// LS Electric XG5000 project: 과년65_2
// PLC NewPLC
// module base 0 slot 0: 입출력 모듈:XBC-DR20S (DC 24V 입력 12점, 릴레이 출력 8점)

PROGRAM NewProgram (task: 스캔 프로그램)

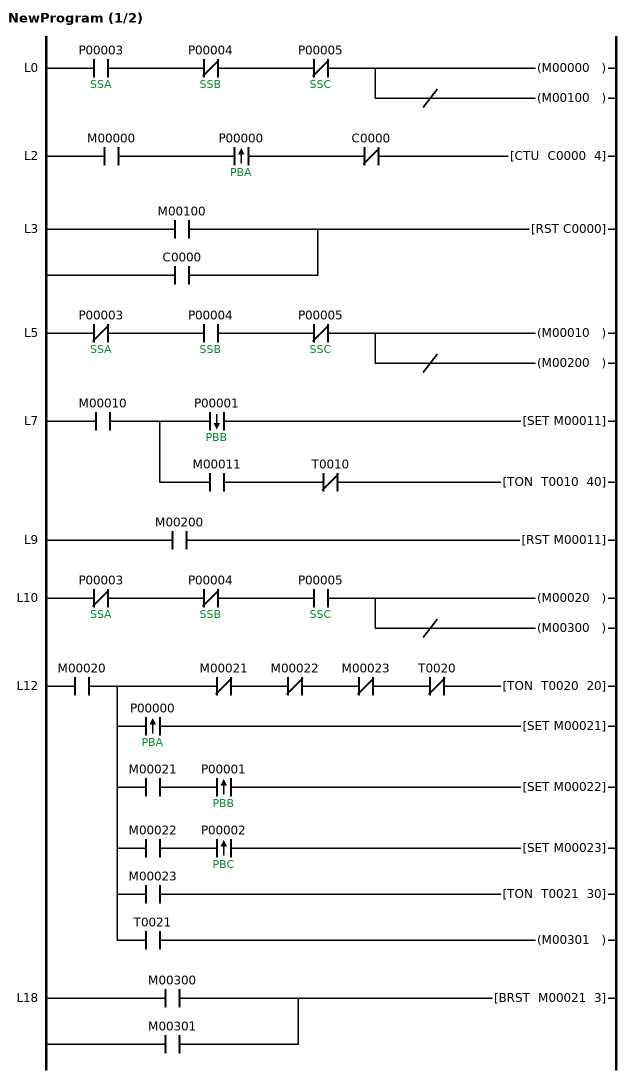
; L0
LOAD      P00003	// SSA
AND NOT   P00004	// SSB
AND NOT   P00005	// SSC
OUT       M00000
NOT
OUT       M00100
; L2
LOAD      M00000
ANDP      P00000	// PBA
AND NOT   C0000
CTU       C0000 4
; L3
LOAD      M00100
OR        C0000
RST       C0000
; L5
LOAD NOT  P00003	// SSA
AND       P00004	// SSB
AND NOT   P00005	// SSC
OUT       M00010
NOT
OUT       M00200
; L7
LOAD      M00010
MPUSH
ANDN      P00001	// PBB
SET       M00011
MPOP
AND       M00011
AND NOT   T0010
TON       T0010 40
; L9
LOAD      M00200
RST       M00011
; L10
LOAD NOT  P00003	// SSA
AND NOT   P00004	// SSB
AND       P00005	// SSC
OUT       M00020
NOT
OUT       M00300
; L12
LOAD      M00020
MPUSH
AND NOT   M00021
AND NOT   M00022
AND NOT   M00023
AND NOT   T0020
TON       T0020 20
MLOAD
ANDP      P00000	// PBA
SET       M00021
MLOAD
AND       M00021
ANDP      P00001	// PBB
SET       M00022
MLOAD
AND       M00022
ANDP      P00002	// PBC
SET       M00023
MLOAD
AND       M00023
TON       T0021 30
MPOP
AND       T0021
OUT       M00301
; L18
LOAD      M00300
OR        M00301
BRST      M00021 3

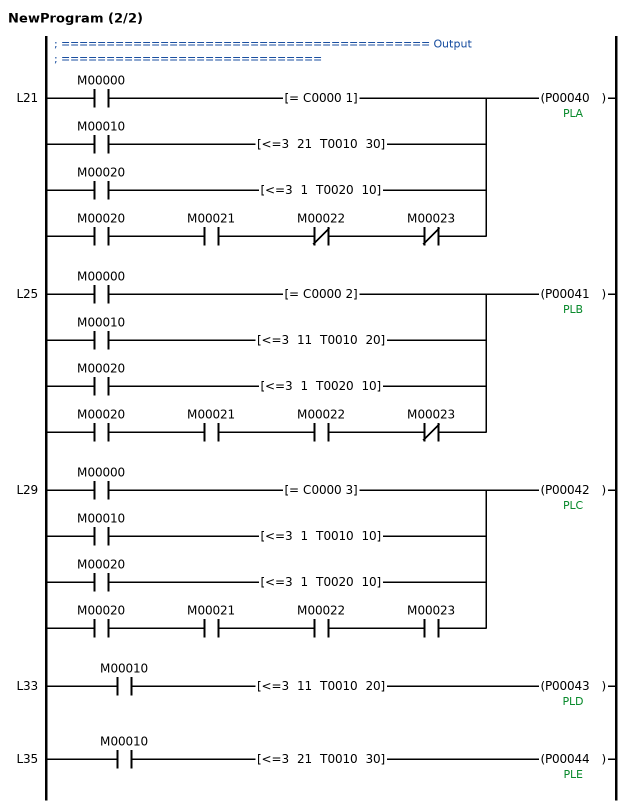
// ========================================= Output =============================
; L21
LOAD      M00000
AND=      C0000 1
LOAD      M00010
AND<=3    21 T0010 30
OR LOAD
LOAD      M00020
AND<=3    1 T0020 10
OR LOAD
LOAD      M00020
AND       M00021
AND NOT   M00022
AND NOT   M00023
OR LOAD
OUT       P00040	// PLA
; L25
LOAD      M00000
AND=      C0000 2
LOAD      M00010
AND<=3    11 T0010 20
OR LOAD
LOAD      M00020
AND<=3    1 T0020 10
OR LOAD
LOAD      M00020
AND       M00021
AND       M00022
AND NOT   M00023
OR LOAD
OUT       P00041	// PLB
; L29
LOAD      M00000
AND=      C0000 3
LOAD      M00010
AND<=3    1 T0010 10
OR LOAD
LOAD      M00020
AND<=3    1 T0020 10
OR LOAD
LOAD      M00020
AND       M00021
AND       M00022
AND       M00023
OR LOAD
OUT       P00042	// PLC
; L33
LOAD      M00010
AND<=3    11 T0010 20
OUT       P00043	// PLD
; L35
LOAD      M00010
AND<=3    21 T0010 30
OUT       P00044	// PLE